FUNCTION TFNextCommandToTilter : INT
VAR_INPUT
	WorkArea : POINTER TO ARRAY [1..MAXAREA] OF TFMachinePalletizer_WorkArea;
	WorkAreaState : POINTER TO ARRAY [1..MAXAREA] OF TFMachinePalletizer_WorkAreaState;
	DistanceFromWAPointer : ARRAY [1..MAXAREA] OF TFMachinePalletizer_WorkAreaSort;
	Forming : POINTER TO ARRAY [1..MAXFORMING] OF TFMachinePalletizer_Forming;
	Mission : POINTER TO TFMachinePalletizer_Mission;
	NextCode : INT;
END_VAR
VAR
	i : INT;
END_VAR

TFNextCommandToTilter := -1;

FOR i:=1 TO MAXAREA DO
	IF WorkArea^[DistanceFromWAPointer[i].cwa].Code = NextCode THEN
		IF WorkArea^[DistanceFromWAPointer[i].cwa].Enable = 1 AND Forming^[WorkAreaState^[DistanceFromWAPointer[i].cwa].F].Enable = 1 AND 
			WorkAreaState^[DistanceFromWAPointer[i].cwa].State = WORKAREA_STATE_OCCUPIED_WORKING THEN
				IF DistanceFromWAPointer[i].cwa = Mission^.PPlace THEN
					TFNextCommandToTilter := Forming^[WorkAreaState^[DistanceFromWAPointer[i].cwa].F].PackXP[WorkAreaState^[DistanceFromWAPointer[i].cwa].P + 1].Grip;
					RETURN;
				ELSE
					TFNextCommandToTilter := Forming^[WorkAreaState^[DistanceFromWAPointer[i].cwa].F].PackXP[WorkAreaState^[DistanceFromWAPointer[i].cwa].P].Grip;
					RETURN;
				END_IF	
		END_IF
	END_IF
END_FOR

END_FUNCTION

(* stored: Version 1.1.0.1, ProductVersion 3.1.4024.11
   POU TFNextCommandToTilter: Id {88cfe9b6-bf9b-4d72-83f6-6135a18daa12}, SpecialFunc None *)
